PROGRAM MAIN
VAR
	bIn : BOOL;
	bOut : BOOL;
	
	iTest : INT;
END_VAR

GVL.bIn := bIn;

GVL.bOut := bOut;



iTest := GVL.iTest;

END_PROGRAM

(* stored: Version 1.1.0.1, ProductVersion 3.1.4024.12
   POU MAIN: Id {3bb257a0-98dd-45b9-85d1-04557b3160eb}, SpecialFunc None *)
